# B&R Automation Studio project WithUpgradesWorking23_08_24 (part 2)

##### ams_rx_msgs.st
```iecst
ACTION msg_ams_000:
	// Status

	// AMS State
	gAMS.status.amsState.0 := ArCanReceive_0.ReceivedFrame.Data[0].0;
	gAMS.status.amsState.1 := ArCanReceive_0.ReceivedFrame.Data[0].1;
	gAMS.status.amsState.2 := ArCanReceive_0.ReceivedFrame.Data[0].2;
	gAMS.status.amsState.3 := ArCanReceive_0.ReceivedFrame.Data[0].3;
	gAMS.status.amsState.4 := ArCanReceive_0.ReceivedFrame.Data[0].4;

	gAMS.status.scEnabled  		:= (gAMS.status.amsStateName = 'SC_ENABLED') OR (gAMS.status.amsStateName = 'TS_ACTIVE') OR (gAMS.status.amsStateName = 'DRIVE');
	gAMS.status.prechargingDone := (gAMS.status.amsStateName = 'TS_ACTIVE') OR (gAMS.status.amsStateName = 'DRIVE');

	// Bank count
	gAMS.status.amsBankCount.0 := ArCanReceive_0.ReceivedFrame.Data[0].5;
	gAMS.status.amsBankCount.1 := ArCanReceive_0.ReceivedFrame.Data[0].6;
	gAMS.status.amsBankCount.2 := ArCanReceive_0.ReceivedFrame.Data[0].7;

	// Error signals
	gAMS.status.error.amsError 				:= ArCanReceive_0.ReceivedFrame.Data[1].0;
	gAMS.status.error.imdError 				:= ArCanReceive_0.ReceivedFrame.Data[1].1;
	gAMS.status.error.hvdcInterlockError 	:= ArCanReceive_0.ReceivedFrame.Data[1].2;
	gAMS.status.error.tempWarn 				:= ArCanReceive_0.ReceivedFrame.Data[1].3;
	gAMS.status.error.voltWarn 				:= ArCanReceive_0.ReceivedFrame.Data[1].4;
	gAMS.status.error.precharge 			:= ArCanReceive_0.ReceivedFrame.Data[1].5;
	gAMS.status.error.airMinus 				:= ArCanReceive_0.ReceivedFrame.Data[1].6;
	gAMS.status.error.airPlus 				:= ArCanReceive_0.ReceivedFrame.Data[1].7;

	// Data
	// gAMS.data.cellVoltageMin_CAN 	:= BYTE_TO_REAL(ArCanReceive_0.ReceivedFrame.Data[2]);
	gAMS.data.cellTempMax 			:= BYTE_TO_REAL(ArCanReceive_0.ReceivedFrame.Data[3]);
	gAMS.data.stateOfCharge 		:= BYTE_TO_REAL(ArCanReceive_0.ReceivedFrame.Data[4]);
	gAMS.status.Counter				:= BYTE_TO_USINT(ArCanReceive_0.ReceivedFrame.Data[5]);
	gAMS.status.RelayError 			:= BYTE_TO_USINT(ArCanReceive_0.ReceivedFrame.Data[6]);

END_ACTION

ACTION msg_ams_011:
	// Cell voltages

	getBankIdAndGroupId;

	//	 Group ID
	//	0	Cell [0-6]
	//	1	Cell [7-13]
	//	2 	Cell [14-20]
	//	3 	Cell [21-27]
	gAMS.status.bank[bankId].cellVoltage[groupId*7 + 0] := BYTE_TO_REAL(ArCanReceive_0.ReceivedFrame.Data[1])*0.02;
	gAMS.status.bank[bankId].cellVoltage[groupId*7 + 1] := BYTE_TO_REAL(ArCanReceive_0.ReceivedFrame.Data[2])*0.02;
	gAMS.status.bank[bankId].cellVoltage[groupId*7 + 2] := BYTE_TO_REAL(ArCanReceive_0.ReceivedFrame.Data[3])*0.02;
	gAMS.status.bank[bankId].cellVoltage[groupId*7 + 3] := BYTE_TO_REAL(ArCanReceive_0.ReceivedFrame.Data[4])*0.02;
	gAMS.status.bank[bankId].cellVoltage[groupId*7 + 4] := BYTE_TO_REAL(ArCanReceive_0.ReceivedFrame.Data[5])*0.02;
	gAMS.status.bank[bankId].cellVoltage[groupId*7 + 5] := BYTE_TO_REAL(ArCanReceive_0.ReceivedFrame.Data[6])*0.02;
	gAMS.status.bank[bankId].cellVoltage[groupId*7 + 6] := BYTE_TO_REAL(ArCanReceive_0.ReceivedFrame.Data[7])*0.02;

END_ACTION

ACTION msg_ams_012:
	// Cell temperatures

	getBankIdAndGroupId;

	// Group Id
	//	0 	Cell [0-4]
	//	1	Cell [5-9]
	gAMS.status.bank[bankId].temperatures[groupId*5 + 0] := BYTE_TO_REAL(ArCanReceive_0.ReceivedFrame.Data[1]);
	gAMS.status.bank[bankId].temperatures[groupId*5 + 1] := BYTE_TO_REAL(ArCanReceive_0.ReceivedFrame.Data[2]);
	gAMS.status.bank[bankId].temperatures[groupId*5 + 2] := BYTE_TO_REAL(ArCanReceive_0.ReceivedFrame.Data[3]);
	gAMS.status.bank[bankId].temperatures[groupId*5 + 3] := BYTE_TO_REAL(ArCanReceive_0.ReceivedFrame.Data[4]);
	gAMS.status.bank[bankId].temperatures[groupId*5 + 4] := BYTE_TO_REAL(ArCanReceive_0.ReceivedFrame.Data[5]); // Changed to 5, was 4 before? May be an error

END_ACTION

ACTION msg_ams_013:
	// Discharge Cell temperatures

	getBankIdAndGroupId;

	// Group Id
	//	0 	Cell [0-6]
	//	1	Cell [7-13]
	gAMS.status.bank[bankId].resistorTemperature[groupId*7 + 0] := BYTE_TO_REAL(ArCanReceive_0.ReceivedFrame.Data[1]);
	gAMS.status.bank[bankId].resistorTemperature[groupId*7 + 1] := BYTE_TO_REAL(ArCanReceive_0.ReceivedFrame.Data[2]);
	gAMS.status.bank[bankId].resistorTemperature[groupId*7 + 2] := BYTE_TO_REAL(ArCanReceive_0.ReceivedFrame.Data[3]);
	gAMS.status.bank[bankId].resistorTemperature[groupId*7 + 3] := BYTE_TO_REAL(ArCanReceive_0.ReceivedFrame.Data[4]);
	gAMS.status.bank[bankId].resistorTemperature[groupId*7 + 4] := BYTE_TO_REAL(ArCanReceive_0.ReceivedFrame.Data[4]);
	gAMS.status.bank[bankId].resistorTemperature[groupId*7 + 5] := BYTE_TO_REAL(ArCanReceive_0.ReceivedFrame.Data[4]);
	gAMS.status.bank[bankId].resistorTemperature[groupId*7 + 6] := BYTE_TO_REAL(ArCanReceive_0.ReceivedFrame.Data[4]);
END_ACTION

ACTION msg_ams_014:
	// Extract first byte which contains the error ID
	errorId := BYTE_TO_USINT(ArCanReceive_0.ReceivedFrame.Data[0]);

	// Reset error timer
	gAMS.status.error.errorTimers[errorId-1](IN := FALSE);
	gAMS.status.error.errorTimers[errorId-1](IN := TRUE);

	//	1  ERROR_AMS_CELL_VOLTAGE_LOW
	//	2  ERROR_AMS_CELL_VOLTAGE_HIGH
	//	3  ERROR_AMS_CELL_TEMP_LOW
	//	4  ERROR_AMS_CELL_TEMP_HIGH
	//	5  ERROR_AMS_LTC6813_COMM
	//	6  ERROR_AMS_SHUNT_COMM
	//	7  ERROR_AMS_UNABLE_TO_OPEN_SC
	//	8  ERROR_AMS_UNABLE_TO_CLOSE_SC
	//	9  ERROR_AMS_UNABLE_TO_OPEN_AIR-
	//	10 ERROR_AMS_UNABLE_TO_CLOSE_AIR-
	//	11 ERROR_AMS_UNABLE_TO_OPEN_AIR+
	//	12 ERROR_AMS_UNABLE_TO_CLOSE_AIR+
	//	13 ERROR_AMS_UNABLE_TO_OPEN_PRE+
	//	14 ERROR_AMS_UNABLE_TO_CLOSE_PRE+
	//	15 ERROR_AMS_PRE_TIMEOUT
	//	16 ERROR_AMS_UNEXPECTED_CHARGE_RATE
	//	17 ERROR_AMS_BANK_COUNT_MISMATCH
	//	18 ERROR_AMS_UNEXSPECPTED_TS_CURRENT
	//	19 ERROR_AMS_RELAY_FAIELD
	//	20 ERROR_AMS_SC_BROKEN
	//	21 AMS_UNFIT_CHARGE_VOLTAGE
	//	22 AMS_MONITOR_ERROR
END_ACTION
```

##### convertData.st
```iecst
ACTION convertData:
	// Takes in data in big endian and converts it to data in litte endian (which is used by the PLC)
	// Switch endian
	dataArr[3] := ArCanReceive_0.ReceivedFrame.Data[2];
	dataArr[2] := ArCanReceive_0.ReceivedFrame.Data[3];
	dataArr[1] := ArCanReceive_0.ReceivedFrame.Data[4];
	dataArr[0] := ArCanReceive_0.ReceivedFrame.Data[5];
	// Extract data from array
	memcpy(ADR(data), ADR(dataArr),4);
END_ACTION
```

##### orion_rx_msgs.st
```iecst
// Frame ID's correspoinding to the orion bms
//  Some message
ACTION msg_orion_001:
	// Byte 0 and 1
	brsmemcpy(ADR(packPower), ADR(ArCanReceive_0.ReceivedFrame.Data[0]), 2 * SIZEOF(ArCanReceive_0.ReceivedFrame.Data[0]));
	gORION.data.packPower 	:= INT_TO_REAL(packPower) / 10; // packpower sent as 0.1kW
	gAMS.data.packPower 	:= gORION.data.packPower;

	// byte 2 and 3, Total pack voltage
	brsmemcpy(ADR(packVoltage), ADR(ArCanReceive_0.ReceivedFrame.Data[2]), 2 * SIZEOF(ArCanReceive_0.ReceivedFrame.Data[2]));
	gAMS.data.batteryVoltage 	:= UINT_TO_REAL(packVoltage) / 10; // Pack voltage sent as 0.1V
	gORION.data.packVoltage 	:= gAMS.data.batteryVoltage;

	// Byte 4 and 5, Total pack Current
	brsmemcpy(ADR(packCurrent), ADR(ArCanReceive_0.ReceivedFrame.Data[4]), 2 * SIZEOF(ArCanReceive_0.ReceivedFrame.Data[4]));
	gAMS.data.outputCurrent 	:= INT_TO_REAL(packCurrent) / 10; // Pack Current sent as 0.1A
	gORION.data.outputCurrent 	:= gAMS.data.outputCurrent;
	gORION.data.chargeCurrent	:= - gAMS.data.outputCurrent;

	// Byte 6 and 7, Charge Current Limit
	brsmemcpy(ADR(gORION.data.CCL), ADR(ArCanReceive_0.ReceivedFrame.Data[6]), 2 * SIZEOF(ArCanReceive_0.ReceivedFrame.Data[6]));

END_ACTION

// Errors and DTC STATUS
ACTION msg_orion_002:
	// BYte 0 and 1
	brsmemcpy(ADR(gAMS.status.DTC1Status), ADR(ArCanReceive_0.ReceivedFrame.Data[0]), 2* SIZEOF(ArCanReceive_0.ReceivedFrame.Data[0]));
	// Byte 2 and 3
	brsmemcpy(ADR(gAMS.status.DTC2Status), ADR(ArCanReceive_0.ReceivedFrame.Data[2]), 2* SIZEOF(ArCanReceive_0.ReceivedFrame.Data[2]));
	gAMS.status.error.highVoltage	:= gAMS.status.DTC1Status.5 OR gAMS.status.DTC2Status.6;
	gAMS.status.error.lowVoltage	:= gAMS.status.DTC1Status.6 OR gAMS.status.DTC2Status.6;
	gAMS.status.error.highTemp 		:= gAMS.status.DTC1Status.7;

	// Byte 4
	// Make some flag wih the MPI to tell the status of these
	gAMS.status.error.imdError 		:= ArCanReceive_0.ReceivedFrame.Data[4].0;
	gAMS.status.error.amsError 		:= ArCanReceive_0.ReceivedFrame.Data[4].1;
	//gAMS.status.error.openSc		:= ArCanReceive_0.ReceivedFrame.Data[4].2;
	gAMS.status.scEnabled			:= ArCanReceive_0.ReceivedFrame.Data[4].2;
	gORION.status.sdcEnabled		:= gAMS.status.scEnabled;
	gAMS.status.relayState.MPEnableSignalStatus := ArCanReceive_0.ReceivedFrame.Data[4].3;

	// BYte 5, rolling counter incrementing every 100ms.
	gORION.data.rollingCounter := BYTE_TO_USINT(ArCanReceive_0.ReceivedFrame.Data[5]);

	// Byte 6 and 7, Discharge Current Limit
	brsmemcpy(ADR(gORION.data.DCL), ADR(ArCanReceive_0.ReceivedFrame.Data[6]), 2 * SIZEOF(ArCanReceive_0.ReceivedFrame.Data[6]));

END_ACTION

ACTION msg_orion_003:
	// 0 and 1, state of relays (Should be sent as little endian)
	brsmemcpy(ADR(gAMS.status.relayState.relayState),ADR(ArCanReceive_0.ReceivedFrame.Data[0]), 2* SIZEOF(ArCanReceive_0.ReceivedFrame.Data[0]));
	gAMS.status.relayState.dischargeRelayEnabled 		:= gAMS.status.relayState.relayState.0;
	gAMS.status.relayState.chargeRelayEnabled	 		:= gAMS.status.relayState.relayState.1;
	gAMS.status.relayState.chargerSafetyEnabled	 		:= gAMS.status.relayState.relayState.2;
	gAMS.status.relayState.malfunctionIndicatorActive 	:= gAMS.status.relayState.relayState.3;
	gAMS.status.relayState.MPI1SignalStatus 			:= gAMS.status.relayState.relayState.4;
	gAMS.status.relayState.alwaysOnSignalStatus 		:= gAMS.status.relayState.relayState.5;
	gAMS.status.relayState.isReadyInputStatus 			:= gAMS.status.relayState.relayState.6;
	gAMS.status.relayState.isChargingInputStatus 		:= gAMS.status.relayState.relayState.7;

	// gAMS.status.relayState.MPI2SignalStatus 			:= gAMS.status.relayState.relayState.8;
	// gAMS.status.relayState.MPI3SignalStatus  		:= gAMS.status.relayState.relayState.9;
	// gAMS.status.relayState.chargeModeStatus 			:= gAMS.status.relayState.relayState.10;
	// gAMS.status.relayState.MPO2SignalStatus 			:= gAMS.status.relayState.relayState.11;
	// gAMS.status.relayState.MPO3SignalStatus 			:= gAMS.status.relayState.relayState.12;
	// gAMS.status.relayState.MPO4SignalStatus 			:= gAMS.status.relayState.relayState.13;
	// gAMS.status.relayState.MPEnableSignalStatus 		:= gAMS.status.relayState.relayState.14;
	// gAMS.status.relayState.MPO1SignalStatus 			:= gAMS.status.relayState.relayState.15;

	// byte 3
	gAMS.data.cellTempMax := BYTE_TO_REAL(ArCanReceive_0.ReceivedFrame.Data[3]); // Max cell temperature of pack, send as (1 degree celcius)
	// Since it is not possible to get all cell voltages independently, max temp i applied to all cells in logic
	appendTemps;

	// Byte 4
	gAMS.data.stateOfCharge := BYTE_TO_REAL(ArCanReceive_0.ReceivedFrame.Data[4]) / 2; // State of charge of battery, (0,5%)

	// Byte 5
	gAMS.status.Counter := BYTE_TO_USINT(ArCanReceive_0.ReceivedFrame.Data[5]); // Counter can be used to make sure Orion BMS is still running and is not stuck

	// byte 6 and 7
	// Failsafe statuses:
	brsmemcpy(ADR(gAMS.status.failsafeStatus.failsafeStatus), ADR(ArCanReceive_0.ReceivedFrame.Data[6]), 2 * SIZEOF(ArCanReceive_0.ReceivedFrame.Data[6]));
	gAMS.status.error.relayFailed := gAMS.status.failsafeStatus.failsafeStatus.2;

END_ACTION

// Related to DCL and CCL in KW
ACTION msg_orion_004:
	// Byte 0-1 Discharge Current limit expressed in KW
	brsmemcpy(ADR(DCL_KW_Temp),ADR(ArCanReceive_0.ReceivedFrame.Data[0]), 2* SIZEOF(ArCanReceive_0.ReceivedFrame.Data[0]));
	gORION.data.DCL_KW := INT_TO_REAL(DCL_KW_Temp)/10; // [0.1kW]

	// Byte 2-3 Charge Current limit expressed in KW
	brsmemcpy(ADR(CCL_KW_Temp),ADR(ArCanReceive_0.ReceivedFrame.Data[2]), 2* SIZEOF(ArCanReceive_0.ReceivedFrame.Data[2]));
	gORION.data.CCL_KW := INT_TO_REAL(CCL_KW_Temp)/10; // [0.1kW]
END_ACTION

 // CELL VOLTAGES, sent though boradcasting
ACTION msg_orion_010:

	// Broadcasted cell voltages from the orion bms
	checksumGiven 		:= BYTE_TO_USINT(ArCanReceive_0.ReceivedFrame.Data[7]);
	checksumCalculated 	:= RX_ORION_ID_BASE + 16#010 + 8;
	checksumCalculated  := checksumCalculated + BYTE_TO_UDINT(ArCanReceive_0.ReceivedFrame.Data[0]);
	checksumCalculated  := checksumCalculated + BYTE_TO_UDINT(ArCanReceive_0.ReceivedFrame.Data[1]);
	checksumCalculated  := checksumCalculated + BYTE_TO_UDINT(ArCanReceive_0.ReceivedFrame.Data[2]);
	checksumCalculated  := checksumCalculated + BYTE_TO_UDINT(ArCanReceive_0.ReceivedFrame.Data[3]);
	checksumCalculated  := checksumCalculated + BYTE_TO_UDINT(ArCanReceive_0.ReceivedFrame.Data[4]);
	checksumCalculated  := checksumCalculated + BYTE_TO_UDINT(ArCanReceive_0.ReceivedFrame.Data[5]);
	checksumCalculated  := checksumCalculated + BYTE_TO_UDINT(ArCanReceive_0.ReceivedFrame.Data[6]);

	brsmemcpy(ADR(checksumValidate),ADR(checksumCalculated),1);

	// Checking if checksum is good
	IF checksumGiven = checksumValidate THEN
		checksumCorrect := checksumCorrect +1;
		// The checksum is correct and data is overwritten
		cellId := BYTE_TO_USINT(ArCanReceive_0.ReceivedFrame.Data[0]);
		brsmemcpy(ADR(tempVoltageHigh), ADR(ArCanReceive_0.ReceivedFrame.Data[1]), SIZEOF(ArCanReceive_0.ReceivedFrame.Data[1]));
		brsmemcpy(ADR(tempVoltageLow), ADR(ArCanReceive_0.ReceivedFrame.Data[2]), SIZEOF(ArCanReceive_0.ReceivedFrame.Data[2]));
		tempVoltage := tempVoltageLow + 256 * tempVoltageHigh;
		gAMS.status.pack.InstantCellVoltage[cellId] := (UINT_TO_REAL(tempVoltage)) / 10000; // recieved data is 2 byte, 0.1mV

		brsmemcpy(ADR(tempVoltageHigh), ADR(ArCanReceive_0.ReceivedFrame.Data[5]), SIZEOF(ArCanReceive_0.ReceivedFrame.Data[5]));
		brsmemcpy(ADR(tempVoltageLow), ADR(ArCanReceive_0.ReceivedFrame.Data[6]), SIZEOF(ArCanReceive_0.ReceivedFrame.Data[6]));
		tempVoltage := tempVoltageLow + 256 * tempVoltageHigh;
		gAMS.status.pack.cellVoltage[cellId] 		:= (UINT_TO_REAL(tempVoltage)) / 10000; // recieved data is 2 byte, 0.1mV

		cellidToBankAndCell;
		gAMS.status.bank[bankId].cellVoltage[bankCellId] := gAMS.status.pack.cellVoltage[cellId];
	END_IF;

END_ACTION

// CELL TEMPERATURES
ACTION msg_orion_011:
	// Broadcasted cell temperatures from the orion bms
	// Is not currently possible to implement
END_ACTION
```

##### shunt_rx_msgs.st
```iecst
ACTION msg_shunt_021:

	// Check if message is of type 'Result' which means it contains measured data and not configuration data
	// If byte 0 is b'0000xxxx' (the 4 msb's are 0) then the type of 'Result'
	IF ArCanReceive_0.ReceivedFrame.Data[0].7 = 0 AND ArCanReceive_0.ReceivedFrame.Data[0].6 = 0 AND
		ArCanReceive_0.ReceivedFrame.Data[0].5 = 0 AND ArCanReceive_0.ReceivedFrame.Data[0].4 = 0 THEN
		// Extract data and switch from big to little endian
		convertData;
		gShunt.data.actCurrent := UDINT_TO_REAL(data)/1000.0; // sent as big indian 4 bytes. [1mA]
	END_IF;

END_ACTION

//Considered to be voltage of the TS side of the car
ACTION msg_shunt_022:
	IF ArCanReceive_0.ReceivedFrame.Data[0].7 = 0 AND ArCanReceive_0.ReceivedFrame.Data[0].6 = 0 AND
		ArCanReceive_0.ReceivedFrame.Data[0].5 = 0 AND ArCanReceive_0.ReceivedFrame.Data[0].4 = 0 THEN
		// Extract data
		convertData;
		gShunt.data.actVoltage := UDINT_TO_REAL(data)/1000.0; // sent as big indian 4 bytes. [1mV]
	END_IF;

END_ACTION

// Not currently in use
ACTION msg_shunt_023:
	IF ArCanReceive_0.ReceivedFrame.Data[0].7 = 0 AND ArCanReceive_0.ReceivedFrame.Data[0].6 = 0 AND
		ArCanReceive_0.ReceivedFrame.Data[0].5 = 0 AND ArCanReceive_0.ReceivedFrame.Data[0].4 = 0 THEN
		// Extract data
		convertData;
		gShunt.data.actVoltage2 := UDINT_TO_REAL(data)/1000.0; // sent as big indian 4 bytes. [1mV]
	END_IF;
END_ACTION

ACTION msg_shunt_026:
	IF ArCanReceive_0.ReceivedFrame.Data[0].7 = 0 AND ArCanReceive_0.ReceivedFrame.Data[0].6 = 0 AND
		ArCanReceive_0.ReceivedFrame.Data[0].5 = 0 AND ArCanReceive_0.ReceivedFrame.Data[0].4 = 0 THEN
		// Extract data
		convertData;
		gShunt.data.actPowerW := UDINT_TO_REAL(data);
		gShunt.data.actPowerKW := gShunt.data.actPowerW/1000.0; // sent as big indian 4 bytes. [1mW]
	END_IF;
END_ACTION

ACTION msg_shunt_027:
	IF ArCanReceive_0.ReceivedFrame.Data[0].7 = 0 AND ArCanReceive_0.ReceivedFrame.Data[0].6 = 0 AND
		ArCanReceive_0.ReceivedFrame.Data[0].5 = 0 AND ArCanReceive_0.ReceivedFrame.Data[0].4 = 0 THEN
		// Extract data
		convertData;
		gShunt.data.actCurrentAS := UDINT_TO_REAL(data);
	END_IF;
END_ACTION

ACTION msg_shunt_028:
	IF ArCanReceive_0.ReceivedFrame.Data[0].7 = 0 AND ArCanReceive_0.ReceivedFrame.Data[0].6 = 0 AND
		ArCanReceive_0.ReceivedFrame.Data[0].5 = 0 AND ArCanReceive_0.ReceivedFrame.Data[0].4 = 0 THEN
		// Extract data
		convertData;
		gShunt.data.actPowerWH  := UDINT_TO_REAL(data);
		gShunt.data.actPowerKWH := gShunt.data.actPowerWH/1000.0;
	END_IF;
END_ACTION
```

### globalDashboard.typ
```iecst
TYPE
	gDashboard_typ : 	STRUCT
		status : gDashboard_status_typ;
		inputs : gDashboard_inputs_typ;
		outputs : gDashboard_outputs_typ;
		cmd : gDashboard_cmd_typ;
		data : gDashboard_data_typ;
	END_STRUCT;
	gDashboard_status_typ : 	STRUCT
		ok : BOOL;
		DashboardDisconnected : BOOL;
		unknownMessageReceived : BOOL;
		unknownMessageID : UDINT;
		timeoutFromDashboard : BOOL;
		canFramesLost : BOOL;
		statusIndex : USINT;
		errorCode : USINT;
	END_STRUCT;
	gDashboard_data_typ : 	STRUCT
		dummy : USINT;
	END_STRUCT;
	gDashboard_inputs_typ : 	STRUCT
		di_buttonSafety : BOOL;
		di_buttonTractive : BOOL;
		di_buttonDrive : BOOL;
		di_button1 : BOOL;
		di_button2 : BOOL;
		di_button3 : BOOL;
		di_button4 : BOOL;
	END_STRUCT;
	gDashboard_cmd_typ : 	STRUCT
		sendVehicleConfigMsg : BOOL;
	END_STRUCT;
	gDashboard_outputs_typ : 	STRUCT
		do_ledTS_OFF : BOOL;
		do_ledIMD : BOOL;
		do_ledAMS : BOOL;
		do_ledEBS : BOOL;
		do_ledREADY : USINT;
		do_ledSC : USINT;
		do_ledLV : BOOL;
		do_ledDV : BOOL;
		Error : USINT;
		com_error_SC : BOOL;
		com_error_Shunt : BOOL;
		com_error_AMS : BOOL;
		com_error_Datalog : BOOL;
		com_error_Dashboard : BOOL;
		com_error_3rd_Inv : BOOL;
		com_error_2nd_Inv : BOOL;
		com_error_1st_Inv : BOOL;
		com_error_0_Inv : BOOL;
		com_error_INS : BOOL;
		com_error_SteeringAngle : BOOL;
		com_error_BreakPressure_Front : BOOL;
		com_error_BreakPressure_Back : BOOL;
		com_error_TorquePedal : BOOL;
		com_error_TorquePedal_Plausi : BOOL;
		com_error_RTDS : BOOL;
		com_error_Cooling : BOOL;
		com_error_LV : BOOL;
		com_error_HighTemperature : BOOL;
	END_STRUCT;
END_TYPE
```

### Program Logical/Dashboard/Dashboard (IEC)

#### Types.typ - Local data types
```iecst
TYPE
	led_states :
		(
		ON,
		OFF,
		BLINKING
		);
END_TYPE
```

#### Variables.var - Local variables
```iecst
VAR
	ledLVState : USINT;
	scLedState : led_states;
	estimatedRange : UINT;
	msgIndex : USINT;
	i : USINT;
	speed : UINT;
	soc : UINT;
	maxTemperature : UINT;
	lvBatVoltage : UINT;
	torqueLimitNm : UINT;
	powerLimitKW : UINT;
	TON_sc : TON;
	ArCanSetBaudrate_0 : ArCanSetBaudrate;
	ArCanSend_0 : ArCanSend;
	ArCanReceive_0 : ArCanReceive;
	communicationState : CAN_STATES;
	deviceName : STRING[127];
	TON_disconnectTimer : TON;
	TON_sendTimer : TON;
	frameIdOffset : UDINT;
	TX_CAN_ID_BASE : {REDUND_UNREPLICABLE} UDINT := 0;
	RX_CAN_ID_BASE : {REDUND_UNREPLICABLE} UDINT := 0;
END_VAR
VAR CONSTANT
	READY_OFF : USINT := 0;
	READY_ON : USINT := 1;
	READY_SLOW_BLINK : USINT := 2;
	READY_FAST_BLINK : USINT := 3;
	SC_OFF : USINT := 0;
	SC_ON : USINT := 1;
	SC_BLINK : USINT := 2;
END_VAR
```

#### ledAMS.st
```iecst
(* Control the AMS LED *)
ACTION ledAMS:
	IF gStateMachine.status.state = STATE_INITIALIZE THEN
		gDashboard.outputs.do_ledAMS := TRUE;
	ELSE
		gDashboard.outputs.do_ledAMS := gAMS.status.error.amsError;
	END_IF;

END_ACTION
```

#### ledSC.st
```iecst
(* Control the SC LED *)

ACTION ledSC:

 	IF gStateMachine.status.state = STATE_INITIALIZE THEN
		gDashboard.outputs.do_ledSC := SC_ON;
	ELSE
		IF gSafetyChain.status.scOK_notEnabled = TRUE AND gSafetyChain.status.scOK = FALSE THEN // If safety chain is OK, but enable button is false change to BLINKING
			gDashboard.outputs.do_ledSC := SC_BLINK;
		ELSIF gSafetyChain.status.scOK = TRUE THEN
			gDashboard.outputs.do_ledSC := SC_ON;
		ELSE
			gDashboard.outputs.do_ledSC := SC_OFF;
		END_IF
	END_IF

END_ACTION
```

#### Send_Bus.st
```iecst
ACTION Send_Bus:

	(* Set timer *)
	TON_sendTimer.PT := T#100ms;
//	TON_sendTimer.PT := T#25ms;

	(* If timer runs out *)
	IF NOT gIsSimulation THEN
		IF TON_sendTimer.Q THEN
			(* Go through each message. Encode and send them *)
			//			FOR i := 0 TO 3 DO
				CASE msgIndex OF
					0: msg_0x000;
					1: msg_0x001;
					2: msg_0x002;
					3: msg_0x003;
					4: msg_0x004;
					ELSE
				END_CASE;
			ArCanSend_0(SendFrame := TRUE);
			ArCanSend_0(SendFrame := FALSE);

			msgIndex := msgIndex + 1;
			IF msgIndex > 4 THEN
				msgIndex := 0;
			END_IF;

//			END_FOR;
			(* Reset timer *)
			TON_sendTimer(IN:=FALSE);
		END_IF;

//		IF gDashboard.cmd.sendVehicleConfigMsg THEN
//			gDashboard.cmd.sendVehicleConfigMsg := FALSE;
//			msg_0x003;
//			ArCanSend_0(SendFrame := TRUE);
//			ArCanSend_0(SendFrame := FALSE);
//		END_IF;

	END_IF;

	(* Start timer *)
	TON_sendTimer(IN:=TRUE);

	ArCanSend_0();
END_ACTION
```

### globalTorqueSensor.typ
```iecst
TYPE
	gTorqueSensor_cmd_typ : 	STRUCT
		torque1 : INT;
		torque2 : INT;
		disablePlausibilityCheck : BOOL;
	END_STRUCT;
	gTorqueSensor_typ : 	STRUCT
		status : gTorqueSensor_status_typ;
		inputs : gTorqueSensor_inputs_typ;
		outputs : gTorqueSensor_outputs_typ;
		data : gTorqueSensor_data_typ;
		cmd : gTorqueSensor_cmd_typ;
	END_STRUCT;
	gTorqueSensor_status_typ : 	STRUCT
		ok : BOOL;
		errorOutOfRangeSensor1 : BOOL;
		errorOutOfRangeSensor2 : BOOL;
		plausibilityError : BOOL;
		torqueEnabled : BOOL;
		torquePercentage : REAL;
		criticalError : BOOL;
		maxTorquePercent : USINT;
	END_STRUCT;
	gTorqueSensor_data_typ : 	STRUCT
		torque1Percent : REAL;
		torque2Percent : REAL;
	END_STRUCT;
	gTorqueSensor_inputs_typ : 	STRUCT
		torque1 : INT;
		torque2 : INT;
	END_STRUCT;
	gTorqueSensor_outputs_typ : 	STRUCT
		dummy : USINT;
	END_STRUCT;
END_TYPE
```

### globalLowVoltageBattery.typ
```iecst
TYPE
	gLowVoltageBattery_typ : 	STRUCT
		status : gLowVoltageBattery_status_typ;
		inputs : gLowVoltageBattery_inputs_typ;
		outputs : gLowVoltageBattery_outputs_typ;
		data : gLowVoltageBattery_data_typ;
	END_STRUCT;
	gLowVoltageBattery_status_typ : 	STRUCT
		full : BOOL;
		empty : BOOL;
		percentageSoc : REAL;
	END_STRUCT;
	gLowVoltageBattery_data_typ : 	STRUCT
		current : REAL;
		voltage : REAL;
	END_STRUCT;
	gLowVoltageBattery_inputs_typ : 	STRUCT
		ai_current : INT;
		ai_voltage : INT;
	END_STRUCT;
	gLowVoltageBattery_outputs_typ : 	STRUCT
		dummy : USINT;
	END_STRUCT;
END_TYPE
```

### globalLowVoltageBattery.var
```iecst
VAR
	gLowVoltageBattery : gLowVoltageBattery_typ;
END_VAR
```

### Program Logical/Sensors/Sensors (IEC)

#### Types.typ - Local data types
```iecst
TYPE
	braking_pedal_variables_typ : 	STRUCT
		brakingPedalFrontMax : UINT;
		brakingPedalFrontMin : UINT;
		brakingPedalRearMax : UINT;
		brakingPedalRearMin : UINT;
		slope : REAL;
	END_STRUCT;
	braking_pedal_constants_typ : 	STRUCT
		frontWarningLimitMaxMax : UINT;
		frontWarningLimitMax : UINT;
		frontWarningLimitMin : UINT;
		frontWarningLimitMinMin : UINT;
		rearWarningLimitMaxMax : UINT;
		rearWarningLimitMax : UINT;
		rearWarningLimitMin : UINT;
		rearWarningLimitMinMin : UINT;
		softBrakingLimit : UINT;
		hardBrakingLimit : UINT;
	END_STRUCT;
	torque_pedal_variables_typ : 	STRUCT
		torquePedalMax2 : UINT;
		torquePedalMax1 : UINT;
		torquePedalMin2 : UINT;
		torquePedalMin1 : UINT;
		TON_torqueOff : TON;
		slope : REAL;
	END_STRUCT;
	torque_pedal_constants_typ : 	STRUCT
		lowLimit2 : UINT;
		highLimit2 : UINT;
		lowLimit1 : UINT;
		highLimit1 : UINT;
		torqueOffUpperHysteresis : REAL;
		torqueOffLowerHysteresis : REAL;
	END_STRUCT;
	steering_angle_constants_typ : 	STRUCT
		highLimit : UINT;
		lowLimit : UINT;
		disconnectionLimit : UINT;
		MAX_ANGLE : REAL;
		MIN_ANGLE : REAL;
	END_STRUCT;
	steering_angle_variables_typ : 	STRUCT
		steeringWheelAngleStr : STRING[80];
		wheelAngleStr : STRING[80];
		leftValue : UINT;
		rightValue : UINT;
	END_STRUCT;
	lv_battery_constants_typ : 	STRUCT
		HighLimit : REAL;
		LowLimit : REAL;
	END_STRUCT;
	lv_battery_variable_typ : 	STRUCT
		TON_batteryEmpty : TON;
		TON_batteryFull : TON;
	END_STRUCT;
END_TYPE
```

#### BrakingPedal.st
```iecst
ACTION BrakingPedalInit:
	(* Sensor limit values *)
	brakingPedalVariables.brakingPedalRearMax 		:= 8000;
	brakingPedalVariables.brakingPedalRearMin 		:= 1655;
	brakingPedalVariables.brakingPedalFrontMax 		:= 8000;
	brakingPedalVariables.brakingPedalFrontMin 		:= 1655;

	(* Braking limits *)
	brakingPedalConstants.hardBrakingLimit			:= 5400;
	brakingPedalConstants.softBrakingLimit			:= 2000;

	(* Upper limit symboling an electrical fault *)
//	brakingPedalConstants.frontWarningLimitMaxMax 	:= brakingPedalVariables.brakingPedalFrontMax + 500;
//	brakingPedalConstants.rearWarningLimitMaxMax 	:= brakingPedalVariables.brakingPedalRearMax  + 500;
	brakingPedalConstants.frontWarningLimitMaxMax 	:= 15250;
	brakingPedalConstants.rearWarningLimitMaxMax 	:= 15250;

	(* Upper limit symboling a mechanical fault *)
	brakingPedalConstants.frontWarningLimitMax 		:= brakingPedalVariables.brakingPedalFrontMax + 100;
	brakingPedalConstants.rearWarningLimitMax 		:= brakingPedalVariables.brakingPedalRearMax  + 100;

	(* Lower limit symboling a mechanical fault *)
	brakingPedalConstants.frontWarningLimitMin 		:= brakingPedalVariables.brakingPedalFrontMin - 100;
	brakingPedalConstants.rearWarningLimitMin 		:= brakingPedalVariables.brakingPedalRearMin  - 100;

	(* Lower limit symboling an electrical fault *)
	brakingPedalConstants.frontWarningLimitMinMin 	:= brakingPedalVariables.brakingPedalFrontMin - 500;
	brakingPedalConstants.rearWarningLimitMinMin 	:= brakingPedalVariables.brakingPedalRearMin  - 500;

END_ACTION

ACTION BrakingPedal:
	(* Detect if brake pedal is being pressed lightly *)
	gBraking.status.softBraking 		 := INT_TO_UINT(gBraking.inputs.ai_brakePressureFront) > brakingPedalConstants.softBrakingLimit OR
											INT_TO_UINT(gBraking.inputs.ai_brakePressureRear)  > brakingPedalConstants.softBrakingLimit OR
											gSoftBrakingForced;

	(* Detect hard braking *)
	gBraking.status.hardBraking 		 := INT_TO_UINT(gBraking.inputs.ai_brakePressureFront) > brakingPedalConstants.hardBrakingLimit OR
										    INT_TO_UINT(gBraking.inputs.ai_brakePressureRear)  > brakingPedalConstants.hardBrakingLimit;

	(* Control brakelight *)
	IF gStateMachine.status.state <> STATE_INITIALIZE THEN
		gBraking.outputs.do_brakeLight   := gBraking.status.softBraking;
	END_IF

	(* Check if brake pressures are out of range *)
	// If brake pressure front get above limit, an error message is shown.
	gBraking.status.errorOutOfRangeFront := INT_TO_UINT(gBraking.inputs.ai_brakePressureFront) >= brakingPedalConstants.frontWarningLimitMax OR
											INT_TO_UINT(gBraking.inputs.ai_brakePressureFront) <= brakingPedalConstants.frontWarningLimitMin;

	// If brake pressure rear get above limit, an error message is shown.
	gBraking.status.errorOutOfRangeRear := 	INT_TO_UINT(gBraking.inputs.ai_brakePressureRear) >= brakingPedalConstants.rearWarningLimitMax OR
											INT_TO_UINT(gBraking.inputs.ai_brakePressureRear) <= brakingPedalConstants.rearWarningLimitMin;

	(* Calculate pedal percentages *)
	IF NOT gBraking.status.errorOutOfRangeFront THEN
		brakingPedalVariables.slope := (100.00)/(UINT_TO_REAL(brakingPedalVariables.brakingPedalFrontMax) - UINT_TO_REAL(brakingPedalVariables.brakingPedalFrontMin));
		gBraking.data.pressurePercentageFront := LIMIT(0 ,brakingPedalVariables.slope * (INT_TO_REAL(gBraking.inputs.ai_brakePressureFront)-UINT_TO_REAL(brakingPedalVariables.brakingPedalFrontMin)),100);
	ELSE
		gBraking.data.pressurePercentageFront := 0;
	END_IF;

	IF NOT gBraking.status.errorOutOfRangeRear THEN
		brakingPedalVariables.slope := (100.00)/(UINT_TO_REAL(brakingPedalVariables.brakingPedalRearMax) - UINT_TO_REAL(brakingPedalVariables.brakingPedalRearMin));
		gBraking.data.pressurePercentageRear := LIMIT(0 ,brakingPedalVariables.slope * (INT_TO_REAL(gBraking.inputs.ai_brakePressureRear)-UINT_TO_REAL(brakingPedalVariables.brakingPedalRearMin)),100);
	ELSE
		gBraking.data.pressurePercentageRear := 0;
	END_IF;

	gBraking.data.pressurePercentage := (gBraking.data.pressurePercentageFront + gBraking.data.pressurePercentageRear)/2.0;

	(* Determine if the brake pedal + sensors are working properly *)
	gBraking.status.ok := NOT gBraking.status.errorOutOfRangeFront AND NOT gBraking.status.errorOutOfRangeRear;

	// Calculate actual pressure
	gBraking.data.pressureBarFront 	:= ((INT_TO_REAL(gBraking.inputs.ai_brakePressureFront)*10/32768)-0.5)*40;
	gBraking.data.pressureBarRear	:= ((INT_TO_REAL(gBraking.inputs.ai_brakePressureRear)*10/32768)-0.5)*40;

END_ACTION
```

#### TorquePedal.st
```iecst
ACTION TorquePedalInit:
	(* Sensor edge values *)
	torquePedalVariables.torquePedalMin1 	:= 13636;
	torquePedalVariables.torquePedalMin2 	:= 2415;
	torquePedalVariables.torquePedalMax1 	:= 21181;
	torquePedalVariables.torquePedalMax2 	:= 7947;

	// Constant for limit torque percent
	IF maxTorquePercentThrottle = 0 THEN
		maxTorquePercentThrottle := 50; // Change to 100, Max Torque Percent
	END_IF;
	gTorqueSensor.status.maxTorquePercent := maxTorquePercentThrottle;

	(* Range for torque sensor 1 *)
	torquePedalConstants.highLimit1 := torquePedalVariables.torquePedalMax1 + 200;
	torquePedalConstants.lowLimit1  := 0;

	(* Range for torque sensor 2 *)
	torquePedalConstants.highLimit2 := torquePedalVariables.torquePedalMax2 + 200;
	torquePedalConstants.lowLimit2 	:= 0;

	(* Torque off hysteresis values *)
	torquePedalConstants.torqueOffUpperHysteresis := 25; // [%]
	torquePedalConstants.torqueOffLowerHysteresis := 5;  // [%]

	(* Plausibility check disable (for test setup) *)
	gTorqueSensor.cmd.disablePlausibilityCheck := FALSE;
END_ACTION

ACTION TorquePedal:
	// Percent of MAX torque at full throttle:
	gTorqueSensor.status.maxTorquePercent := maxTorquePercentThrottle;

	gTorqueSensor.status.errorOutOfRangeSensor1 := 	INT_TO_UINT(gTorqueSensor.inputs.torque1) > torquePedalConstants.highLimit1 OR
													INT_TO_UINT(gTorqueSensor.inputs.torque1) < torquePedalConstants.lowLimit1;

	gTorqueSensor.status.errorOutOfRangeSensor2 := 	INT_TO_UINT(gTorqueSensor.inputs.torque2) > torquePedalConstants.highLimit2 OR
													INT_TO_UINT(gTorqueSensor.inputs.torque2) < torquePedalConstants.lowLimit2;

	(* Calculate pedal percentages *)

	// Sensor 1
	IF NOT gTorqueSensor.status.errorOutOfRangeSensor1 THEN
		torquePedalVariables.slope := (100)/(UINT_TO_REAL(torquePedalVariables.torquePedalMax1) - UINT_TO_REAL(torquePedalVariables.torquePedalMin1));
		gTorqueSensor.data.torque1Percent := LIMIT(0 ,torquePedalVariables.slope * (INT_TO_REAL(gTorqueSensor.inputs.torque1)-(10+UINT_TO_REAL(torquePedalVariables.torquePedalMin1))),100);
	ELSE
		gTorqueSensor.data.torque1Percent := 0;
	END_IF;
	// gTorqueSensor.status.maxTorquePercent TODO: USE THIS FOR SCALING
	// Sensor 2
	IF NOT gTorqueSensor.status.errorOutOfRangeSensor2 THEN
		torquePedalVariables.slope := (100)/(UINT_TO_REAL(torquePedalVariables.torquePedalMax2) - UINT_TO_REAL(torquePedalVariables.torquePedalMin2));
		gTorqueSensor.data.torque2Percent := LIMIT(0 ,torquePedalVariables.slope * (INT_TO_REAL(gTorqueSensor.inputs.torque2)-UINT_TO_REAL(torquePedalVariables.torquePedalMin2)),100);
	ELSE
		gTorqueSensor.data.torque2Percent := 0;
	END_IF;

	// Sensor 1 is arbitrarily taken to be the torque percentage
	// Value is then scaled by desired power
	gTorqueSensor.status.torquePercentage := gTorqueSensor.data.torque1Percent*gTorqueSensor.status.maxTorquePercent/100;

	(* Test if torque sensor values are out of range of each other*)
	TorqueSensorsOutOfRange;
	TorqueOff;

	(* Report critical error if either of the torque pedal sensors leave their working range *)
	gTorqueSensor.status.criticalError := gTorqueSensor.status.errorOutOfRangeSensor1 OR gTorqueSensor.status.errorOutOfRangeSensor2 OR gTorqueSensor.status.plausibilityError;

	(* Determine if the torque pedal is working properly *)
	gTorqueSensor.status.ok := NOT gTorqueSensor.status.criticalError;

END_ACTION

(* Test if torque pedals are more than 10% different than each other *)
ACTION TorqueSensorsOutOfRange:
	IF gTorqueSensor.cmd.disablePlausibilityCheck THEN
		gTorqueSensor.status.plausibilityError := FALSE;
	ELSE
		// check if torque sensor 1 and 2 vary more than 5 %
		gTorqueSensor.status.plausibilityError := ABS(gTorqueSensor.data.torque1Percent - gTorqueSensor.data.torque2Percent) > 5;
	END_IF;
END_ACTION

ACTION TorqueOff:
	IF gTorqueSensor.status.torqueEnabled THEN
		(* Test the criterias for turning off the torque. If they are met start timer *)
		IF 	gBraking.status.softBraking AND
			(gTorqueSensor.data.torque1Percent >= torquePedalConstants.torqueOffUpperHysteresis OR
			 gTorqueSensor.data.torque2Percent >= torquePedalConstants.torqueOffUpperHysteresis OR
		 	 gORION.data.packPower >= 5.0) THEN

			torquePedalVariables.TON_torqueOff.PT := T#250ms;	// Set timer duration TODO: Change to 500 that is the limit in the rules
			torquePedalVariables.TON_torqueOff.IN := TRUE;		// Start timer
		ELSE
			torquePedalVariables.TON_torqueOff.IN := FALSE;		// Else stop timer
		END_IF

		IF torquePedalVariables.TON_torqueOff.Q THEN			// If timer runs out
			gTorqueSensor.status.torqueEnabled := FALSE;		// Remove torque
		ELSE
			gTorqueSensor.status.torqueEnabled := TRUE;			// Else keep torque
		END_IF;
	ELSE
		(* Test the criterias for turning on the torque *)
		gTorqueSensor.status.torqueEnabled := 	gTorqueSensor.data.torque1Percent < torquePedalConstants.torqueOffLowerHysteresis AND
												gTorqueSensor.data.torque2Percent < torquePedalConstants.torqueOffLowerHysteresis AND (NOT gBraking.status.softBraking);
		torquePedalVariables.TON_torqueOff.IN := FALSE;			// Make sure the torque timer is stopped
	END_IF
	torquePedalVariables.TON_torqueOff();						// Run torque timer
END_ACTION
```

#### LowVoltageBattery.st
```iecst
ACTION LowVoltageBatteryInit:
	lvBatteryConstants.HighLimit := 13.0;
	lvBatteryConstants.LowLimit  := 11.0;

	lvBatteryVariables.TON_batteryEmpty.PT := T#1s;
	lvBatteryVariables.TON_batteryFull.PT := T#1s;
END_ACTION

ACTION LowVoltageBattery:
//	gLowVoltageBattery.data.lowVoltageBatteryVoltage :=  0.001209 * gLowVoltageBattery.inputs.im_LowVoltageBattery_Voltage + 0.6351;
	gLowVoltageBattery.data.voltage :=  (32.0/32767.0) * gLowVoltageBattery.inputs.ai_voltage;

	gLowVoltageBattery.data.current := (((10.0/32767.0)*gLowVoltageBattery.inputs.ai_current) - 0.5)/0.08;

	// Check if the low voltage battery is below a threshold and set status flag
	lvBatteryVariables.TON_batteryEmpty(IN := gLowVoltageBattery.data.voltage < lvBatteryConstants.LowLimit);
	gLowVoltageBattery.status.empty := lvBatteryVariables.TON_batteryEmpty.Q;

	// Check of the low voltage battery is above a threshold and set status flag
	lvBatteryVariables.TON_batteryFull(IN := gLowVoltageBattery.data.voltage > lvBatteryConstants.HighLimit);
	gLowVoltageBattery.status.full := lvBatteryVariables.TON_batteryFull.Q;

END_ACTION
```

### globalSensorNet.var
```iecst
VAR
	gSensorNet : gSensorNet_typ;
END_VAR
VAR CONSTANT
	SENSOR_NET_POLY_LEN : USINT := 8; (*Length - 1. Writing 8 here means its a 9th order polynomial*)
END_VAR
```

### Program Logical/SensorNet/globalSensorNet

#### Main.st
```iecst
PROGRAM _INIT
	(* Insert code here *)

END_PROGRAM

PROGRAM _CYCLIC

	calculateSensorNetOut_0(input := gSensorNet.data.coolingTemp1.input, polyCoeffs := gSensorNet.data.coolingTemp1.polyCoeffs);
	gSensorNet.data.coolingTemp1.value := calculateSensorNetOut_0.output;

END_PROGRAM

PROGRAM _EXIT
	(* Insert code here *)

END_PROGRAM
```

### globalRTDS.var
```iecst
VAR
	gRTDS : gRTDS_typ;
END_VAR
```

### Program Logical/Actuators/Output (IEC)

#### Types.typ - Local data types
```iecst
TYPE
	rtdsVariables_typ : 	STRUCT
		TON_RTDS : TON;
	END_STRUCT;
	rtdsConstants_typ : 	STRUCT
		RTDSCurrent : INT;
	END_STRUCT;
END_TYPE
```

#### Variables.var - Local variables
```iecst
VAR
	i : USINT;
	rtdsVariables : rtdsVariables_typ;
	rtdsConstants : rtdsConstants_typ;
END_VAR
```

### globalCooling.typ
```iecst
TYPE
	gCooling_typ : 	STRUCT
		outputs : gCooling_outputs_typ;
		inputs : gCooling_inputs_typ;
		data : gCooling_data_typ;
		cmd : gCooling_cmd_typ;
		status : gCooling_status_typ;
	END_STRUCT;
	gCooling_outputs_typ : 	STRUCT
		do_fan : ARRAY[0..NUMBER_OF_FANS]OF BOOL;
		do_pump : ARRAY[0..NUMBER_OF_PUMPS]OF BOOL;
	END_STRUCT;
	gCooling_inputs_typ : 	STRUCT
		ai_coolingTemp : ARRAY[0..NUMBER_OF_COOLING_SENSORS]OF INT;
		im_pumpCurrent : ARRAY[0..NUMBER_OF_PUMPS]OF INT;
	END_STRUCT;
	gCooling_cmd_typ : 	STRUCT
		manualMode : BOOL;
		inverterMaxTemp : REAL;
		motorMaxTemp : REAL;
	END_STRUCT;
	gCooling_status_typ : 	STRUCT
		ok : BOOL;
		error : BOOL;
		pumpError : ARRAY[0..1]OF BOOL;
		pumpState : ARRAY[0..1]OF PUMP_STATES;
		warningHighTemperature : BOOL;
		warningInverterHighTemp : BOOL;
		warningMotorHighTemp : BOOL;
	END_STRUCT;
	gCooling_data_typ : 	STRUCT
		coolingSysTemp : ARRAY[0..NUMBER_OF_COOLING_SENSORS]OF REAL;
	END_STRUCT;
	PUMP_STATES :
		(
		PUMP_STATE_OK,
		PUMP_STATE_NO_WATER,
		PUMP_STATE_NOT_CONNECTED
		);
END_TYPE
```

### globalCooling.var
```iecst
VAR CONSTANT
	NUMBER_OF_FANS : USINT := 2;
	NUMBER_OF_COOLING_SENSORS : USINT := 2;
	NUMBER_OF_PUMPS : USINT := 2;
END_VAR
VAR
	gCooling : gCooling_typ;
END_VAR
```

### globalINS.typ
```iecst
TYPE
	gINS_status_typ : 	STRUCT
		ok : BOOL;
	END_STRUCT;
	gINS_data_typ : 	STRUCT
		actLonVelocity_ms : REAL;
		actLatVelocity_ms : REAL;
		actLonVelocity_kmh : REAL;
		actLatVelocity_kmh : REAL;
		actLonAcceleration : REAL;
		actLatAcceleration : REAL;
		actYawRate : REAL;
		actDistTraveledKm : REAL;
		actDistTraveledM : REAL;
		distEstimated : REAL;
	END_STRUCT;
	gINS_input_typ : 	STRUCT
		gyroX : REAL;
		gyroY : REAL;
		gyroZ : REAL;
		accX : REAL;
		accY : REAL;
		accZ : REAL;
		velX : REAL;
		velY : REAL;
		velZ : REAL;
	END_STRUCT;
	gINS_typ : 	STRUCT
		data : gINS_data_typ;
		status : gINS_status_typ;
		input : gINS_input_typ;
	END_STRUCT;
END_TYPE
```

### Program Logical/INS/INS (IEC)

#### Variables.var - Local variables
```iecst
VAR
	messageOk : BOOL;
	distDelta : REAL;
	cycletime : UDINT;
	RTInfo_0 : RTInfo;
	Receiver : Receiver_typ := (0); (*local Struktur with all instances and variables*)
END_VAR
VAR CONSTANT
	BUSY : UINT := 65535; (*Functionblock BUSY status*)
END_VAR
VAR
	socActual : REAL;
	socPrevious : REAL;
	distActual : REAL;
	distPrevious : REAL;
	MTFilterMovingAverage_0 : MTFilterMovingAverage;
	TON_rangEstTimer : TON;
END_VAR
```

#### extractInsData.st
```iecst
(* Action to pick out data for each variable from the received INS data *)
ACTION extractInsData:

	// Byte 0-5: Header

	// Data

	// 6 - 9: AccX
	memcpy(ADR(gINS.input.accX), ADR(Receiver.receive_data)+6,4);
	// 10-13: AccY
	memcpy(ADR(gINS.input.accY), ADR(Receiver.receive_data)+10,4);
	// 14-17: AccZ
	memcpy(ADR(gINS.input.accZ), ADR(Receiver.receive_data)+14,4);

	// 18-21: GyroX
	memcpy(ADR(gINS.input.gyroX), ADR(Receiver.receive_data)+18,4);
	// 22-25: GyroY
	memcpy(ADR(gINS.input.gyroY), ADR(Receiver.receive_data)+22,4);
	// 26-29: GyroZ
	memcpy(ADR(gINS.input.gyroZ), ADR(Receiver.receive_data)+26,4);

	// 30-33: VelX
	memcpy(ADR(gINS.input.velX), ADR(Receiver.receive_data)+30,4);
	// 34-37: VelY
	memcpy(ADR(gINS.input.velY), ADR(Receiver.receive_data)+34,4);
	// 38-41: VelZ
	memcpy(ADR(gINS.input.velZ), ADR(Receiver.receive_data)+38,4);

	// 42-42: Checksum / CRC

END_ACTION
```

#### rangeEst.st
```iecst
ACTION rangeEstimation:
	(* Handle timer *)
	TON_rangEstTimer.IN := TRUE;
	TON_rangEstTimer();

	socActual 	:= gAMS.data.stateOfCharge;
	distActual 	:= gINS.data.actDistTraveledKm;

	(* If timeout occurs *)
	IF TON_rangEstTimer.Q THEN
		(* Reset Timer *)
		TON_rangEstTimer(IN := FALSE);
		(* if the previous SoC is higher *)
		IF socActual < socPrevious THEN
			(* Calculate next value in range estimation *)
			MTFilterMovingAverage_0(In := LIMIT(0,distPrevious - (socPrevious*(distActual-distPrevious))/(socActual-socPrevious),50));
			gINS.data.distEstimated := MTFilterMovingAverage_0.Out;
			(* Previous SoC is lower than new, indication of charging *)
		END_IF;
		distPrevious := gINS.data.actDistTraveledKm;
		socPrevious  := gAMS.data.stateOfCharge;
	END_IF;
END_ACTION
```

#### distMeas.st
```iecst
ACTION distanceMeasurement:

	// dt = cycletime
	// h = ms/(1000*60*60) => h = ms/(3600000)
	distDelta := gINS.data.actLonVelocity_kmh * (UDINT_TO_REAL(cycletime)/3600000.0);

	// Increment distance traveled by distance delta
	gINS.data.actDistTraveledKm := gINS.data.actDistTraveledKm + distDelta;

	// Calculate the distance in meters as well
	gINS.data.actDistTraveledM := gINS.data.actDistTraveledKm*1000.0;

END_ACTION
```

#### checkMessageValidity.st
```iecst
ACTION checkMessageValidity:
	messageOk := TRUE;
END_ACTION
```

### Program Logical/Misc/DataLogging/DataLog

#### Types.typ
```iecst
TYPE
	this_typ : 	STRUCT
		state : UINT;
		tmpStr : STRING[80];
		idxStr : STRING[10];
		strIdxPos : DINT;
		csvData : ARRAY[0..DATALOG_MAX_LOG_VARS]OF STRING[200];
		fileInfoSetting : fiFILE_INFO;
		DTGetTime_0 : DTGetTime;
		header : MpRecipeXmlHeaderType;
		MpDataRegPar : ARRAY[0..DATALOG_MAX_MAPP_VARS]OF MpDataRegPar;
		timestamp : this_timestamp_typ;
		pvData : ARRAY[0..DATALOG_MAX_LOG_VARS]OF this_pvdata_typ;
		pvRegData : ARRAY[0..DATALOG_MAX_MAPP_VARS]OF this_pvRegData_typ;
		okToRestart : BOOL;
		TON_errorReset : TON;
		TON_recordDelay : TON;
		systemReadyToLog : BOOL;
		maxIdxVariableX : USINT;
		brdkUSBConnect_0 : brdkUSBConnect;
		FileCreate_0 : FileCreate;
	END_STRUCT;
	this_timestamp_typ : 	STRUCT
		str : STRING[64];
		old : DATE_AND_TIME;
	END_STRUCT;
	this_pvdata_typ : 	STRUCT
		variable : STRING[200];
		enableVar : STRING[200];
	END_STRUCT;
	this_pvRegData_typ : 	STRUCT
		variable : STRING[100];
		enableVar : STRING[100];
		enable : BOOL;
		address : UDINT;
		datalength : UDINT;
	END_STRUCT;
END_TYPE
```

#### Variables.var
```iecst
VAR
	this : this_typ;
	i : UINT;
	j : USINT;
	pBool : REFERENCE TO BOOL; (*Temp pointer to bool*)
	noOfPvVars : UINT;
	MpDataRecorder_0 : MpDataRecorder;
	MpDataRecorderConfig_0 : MpDataRecorderConfig;
	MpDataRecorderConfiguration : MpDataRecorderConfigType;
	MpRecipeCsv_0 : MpRecipeCsv;
	MpRecipeRegPar_csv : MpRecipeRegPar;
	FileInfo_0 : FileInfo;
	DirCreate_0 : DirCreate;
	RTInfo_0 : RTInfo;
END_VAR
```

#### DataLog.st
```iecst
PROGRAM _INIT

	RTInfo_0(enable := TRUE);
	initSetup;

END_PROGRAM

PROGRAM _CYCLIC
	// call actions
	setup;

	//detect if config.enable is changed then restart datalog
	FOR i:=0 TO DATALOG_MAX_MAPP_VARS DO
		IF this.okToRestart AND this.pvRegData[i].variable <> '' THEN
			IF this.pvRegData[i].address <> 0 AND this.pvRegData[i].datalength = 1 THEN
				pBool ACCESS this.pvRegData[i].address;
				IF pBool <> this.pvRegData[i].enable THEN
					this.state := 0; //restart
				END_IF
			END_IF
		ELSE EXIT;
		END_IF
	END_FOR

	//if file is changed then restart datalog
	FileInfo_0();
	IF this.okToRestart AND this.timestamp.old <> this.fileInfoSetting.modTime THEN
		this.state := 0; //restart
	END_IF

	CASE this.state OF
		0:	// wait for connected usb device
			IF this.brdkUSBConnect_0.status = BRDK_USB_STATUS_FB_READY THEN
				// finds the first available node
				FOR i := 0 TO BRDK_USB_MAX_DEVICES-1 DO
					IF this.brdkUSBConnect_0.node[i].device <> '' THEN
						this.FileCreate_0.pDevice	:= ADR(this.brdkUSBConnect_0.node[i].device);
						this.state := 5;
					END_IF
				END_FOR
			END_IF

		5: //create log folder
			this.okToRestart := FALSE;
			this.timestamp.old := this.fileInfoSetting.modTime;
			MpDataRecorder_0.Enable := FALSE;
			DirCreate_0.enable := TRUE;
			IF DirCreate_0.status = fiERR_DIR_ALREADY_EXIST THEN
				DirCreate_0.enable := FALSE;
				this.state := 10;
			END_IF
			DirCreate_0();

		10:
			MpRecipeRegPar_csv.Enable := TRUE;
			IF MpRecipeRegPar_csv.Active THEN
				this.state := 20;
			ELSIF MpRecipeRegPar_csv.Error THEN
				this.state := 65000;
			END_IF

		20:
			MpRecipeCsv_0.Enable := TRUE;
			IF MpRecipeCsv_0.Active THEN
				this.state := 30;
			ELSIF MpRecipeCsv_0.Error THEN
				this.state := 65000;
			END_IF

		30: //DatalogSettings.csv ok?
			IF FileInfo_0.status = ERR_OK THEN
				this.state := 40;
			ELSIF FileInfo_0.status = fiERR_FILE_NOT_FOUND THEN
				this.state := 300;
			ELSIF FileInfo_0.status = ERR_FUB_BUSY THEN
			ELSE
				this.state := 65000;
			END_IF

		40:
			MpRecipeCsv_0.Load := TRUE;
			IF MpRecipeCsv_0.CommandDone THEN
				MpRecipeCsv_0.Load := FALSE;
				this.state := 45;
			ELSIF MpRecipeCsv_0.Error THEN
				this.state := 65000;
			END_IF

		45:
			MpDataRecorder_0.Enable := TRUE;
			IF MpDataRecorder_0.Active THEN
				this.state := 50;
			ELSIF MpDataRecorder_0.Error THEN
				this.state := 65000;
			END_IF

		50://find logVar#logVarEnable and split it
			brsmemset(ADR(this.pvRegData), 0, SIZEOF(this.pvRegData));
			brsmemset(ADR(this.pvData), 0, SIZEOF(this.pvData));
			FOR i:=0 TO DATALOG_MAX_LOG_VARS DO
				IF gDataLogging.data.csvData[i] <> '' THEN
					this.strIdxPos := brdkStrSearch(ADR(gDataLogging.data.csvData[i]),ADR('#'));
					IF this.strIdxPos > 0 THEN //enable/disable variable found
						this.pvData[i].variable 	:= gDataLogging.data.csvData[i];
						this.pvData[i].enableVar 	:= gDataLogging.data.csvData[i];
						brdkStrSlice(ADR(this.pvData[i].variable), 0, this.strIdxPos);
						brdkStrSlice(ADR(this.pvData[i].enableVar), this.strIdxPos+1, SIZEOF(this.pvData[i].enableVar));
					ELSE
						this.pvData[i].variable := gDataLogging.data.csvData[i];
					END_IF
				ELSE EXIT;
				END_IF
			END_FOR
			this.state := 60;

		60://find and replace [x]. to [0..this.maxIdxVariableX]
			noOfPvVars := 0;
			FOR i:=0 TO DATALOG_MAX_LOG_VARS DO
				IF gDataLogging.data.csvData[i] <> '' THEN
					this.strIdxPos := brdkStrSearch(ADR(this.pvData[i].variable), ADR('[x]'));
				 	IF this.strIdxPos > 0 THEN
				 		FOR j:=0 TO this.maxIdxVariableX DO
							this.tmpStr := '[x]';
							brsitoa(j, ADR(this.idxStr));
							brdkStrReplace(ADR(this.tmpStr), ADR('x'), ADR(this.idxStr));
							this.pvRegData[noOfPvVars].variable 	:= this.pvData[i].variable;
							this.pvRegData[noOfPvVars].enableVar 	:= this.pvData[i].enableVar;
							brdkStrReplace(ADR(this.pvRegData[noOfPvVars].variable), ADR('[x]'), ADR(this.tmpStr));
							brdkStrReplace(ADR(this.pvRegData[noOfPvVars].enableVar), ADR('[x]'), ADR(this.tmpStr));
							PV_xgetadr(ADR(this.pvRegData[noOfPvVars].enableVar), ADR(this.pvRegData[noOfPvVars].address), ADR(this.pvRegData[noOfPvVars].datalength));
							noOfPvVars := noOfPvVars + 1;
						END_FOR
					ELSE
						this.pvRegData[noOfPvVars].variable 	:= this.pvData[i].variable;
						this.pvRegData[noOfPvVars].enableVar 	:= this.pvData[i].enableVar;
						PV_xgetadr(ADR(this.pvRegData[noOfPvVars].enableVar), ADR(this.pvRegData[noOfPvVars].address), ADR(this.pvRegData[noOfPvVars].datalength));
						noOfPvVars := noOfPvVars + 1;
				 	END_IF
				ELSE EXIT;
				END_IF
			END_FOR
			this.state := 65;

		65: //clear all reg pars before init again
			FOR i:=0 TO DATALOG_MAX_MAPP_VARS DO
				this.MpDataRegPar[i].Enable := FALSE;
			END_FOR
			this.state := 70;

		70: //registre pv's
			FOR i:=0 TO DATALOG_MAX_MAPP_VARS DO
				IF this.pvRegData[i].variable <> '' THEN
					this.MpDataRegPar[i].MpLink 		:= ADR(gDataRecorder);
					this.MpDataRegPar[i].Description 	:= ADR(this.pvRegData[i].variable);
					this.MpDataRegPar[i].PVName			:= ADR(this.pvRegData[i].variable);
					IF this.pvRegData[i].address <> 0 AND this.pvRegData[i].datalength = 1 THEN
						pBool ACCESS this.pvRegData[i].address;
						this.pvRegData[i].enable := pBool;
					ELSE
						this.pvRegData[i].enable := TRUE;
					END_IF
					this.MpDataRegPar[i].Enable	:= this.pvRegData[i].enable;
				ELSE EXIT;
				END_IF
			END_FOR
			this.okToRestart := TRUE;
			this.state := 80;

		80: //wait for system up and running
			IF this.systemReadyToLog THEN
				MpDataRecorder_0.Enable := TRUE;
				this.state := 85;
			END_IF

		85: //active
			IF MpDataRecorder_0.Active THEN
				this.TON_recordDelay.IN := TRUE;
				this.state := 90;
			ELSIF MpDataRecorder_0.Error THEN
				this.state := 65000;
			END_IF

		90: //delay before start recording
			IF this.TON_recordDelay.Q THEN
				this.TON_recordDelay.IN := FALSE;
				MpDataRecorder_0.Record := TRUE;
				this.state := 100;
			END_IF

		100: //ready
			gDataLogging.status.dataloggingActive := TRUE;
			IF gCreateLogFile THEN
				this.okToRestart := FALSE;
				MpDataRecorder_0.SnapShot := TRUE;
				this.state := 110;
			ELSIF NOT MpDataRecorder_0.Enable THEN // restart after download
				gCreateLogFile := FALSE;
				this.state := 0;
			ELSIF MpDataRecorder_0.Error THEN
				gCreateLogFile := FALSE;
				this.state := 65000;
			END_IF

			IF MpDataRecorder_0.Info.CurrentFileSize > 900 THEN
				this.state := 5;
			END_IF

		110: //waiting for datalog file created
			IF MpDataRecorder_0.SnapShotDone THEN
				MpDataRecorder_0.SnapShot 	:= FALSE;
				gCreateLogFile 				:= FALSE;
				this.state 					:= 100;
			ELSIF MpDataRecorder_0.Error THEN
				MpDataRecorder_0.ErrorReset	:= TRUE;
				MpDataRecorder_0.SnapShot 	:= FALSE;
				gCreateLogFile 				:= FALSE;
				this.state 					:= 65000;
			END_IF

		300: //create DatalogSettings.csv
			MpRecipeCsv_0.Save := TRUE;
			IF MpRecipeCsv_0.CommandDone THEN
				MpRecipeCsv_0.Save := FALSE;
				this.state := 0;
			ELSIF MpRecipeCsv_0.Error THEN
				this.state := 65000;
			END_IF

		65000://ERROR HANDLING = NONE :/
			this.TON_errorReset.IN	:= TRUE;
			IF this.TON_errorReset.Q THEN
				this.TON_errorReset.IN		:= FALSE;
				MpDataRecorder_0.Enable 	:= FALSE;
				MpRecipeRegPar_csv.Enable 	:= FALSE;
				MpRecipeCsv_0.Enable		:= FALSE;
				FileInfo_0.enable			:= FALSE;
				this.state					:= 0;
			END_IF

	END_CASE

	// Function Block Calls
	this.TON_errorReset(PT := T#10s);

	IF this.state <> 100 OR this.brdkUSBConnect_0.status <> BRDK_USB_STATUS_FB_READY THEN
		gDataLogging.status.dataloggingActive := FALSE;
	END_IF

	this.TON_recordDelay();
	IF MpDataRecorder_0.Active THEN
		FOR i:=0 TO DATALOG_MAX_MAPP_VARS DO
			this.MpDataRegPar[i]();
		END_FOR
	END_IF
	MpDataRecorderConfig_0();
	MpDataRecorder_0();
	MpRecipeRegPar_csv();
	MpRecipeCsv_0();
	this.brdkUSBConnect_0();

END_PROGRAM

PROGRAM _EXIT
	// Disable Mapp Function Blocks
	MpDataRecorder_0(Enable := FALSE);
	MpDataRecorderConfig_0(Enable := FALSE);
	MpRecipeCsv_0(Enable := FALSE);
	MpRecipeRegPar_csv(Enable := FALSE);
END_PROGRAM
```

#### setup.st
```iecst
ACTION setup:
	IF this.brdkUSBConnect_0.node[0].device <> '' THEN
		MpRecipeRegPar_csv.MpLink 	:= ADR(gRecipeCsv);
		MpRecipeRegPar_csv.PVName 	:= ADR('DataLog:gDataLogging.inputs.csvData');
		MpRecipeRegPar_csv.Category	:= ADR('datalogSettings');

		MpRecipeCsv_0.MpLink 		:= ADR(gRecipeCsv);
		MpRecipeCsv_0.DeviceName 	:= ADR(this.brdkUSBConnect_0.node[0].device);
		MpRecipeCsv_0.FileName 		:= ADR('log/DatalogSettings');
		MpRecipeCsv_0.Category		:= ADR('datalogSettings');

		MpDataRecorder_0.MpLink			:= ADR(gDataRecorder);
		MpDataRecorder_0.DeviceName		:= ADR(this.brdkUSBConnect_0.node[0].device);
		MpDataRecorder_0.RecordMode 	:= mpDATA_RECORD_MODE_TIME;
		MpDataRecorder_0.SamplingTime	:= RTInfo_0.cycle_time / 1000; //micro to milli

		MpDataRecorderConfiguration.DecimalDigits	:= 3;
		MpDataRecorderConfiguration.BufferSize		:= 50000; //kB
		MpDataRecorderConfiguration.PowerFailSafe	:= FALSE;
		MpDataRecorderConfiguration.FileNamePattern	:= 'Datalog_%Y%m%d_%H%M%S.csv';
		MpDataRecorderConfiguration.DecimalMark		:= '.';
		MpDataRecorderConfiguration.AutoSave		:= FALSE;

		MpDataRecorderConfig_0.MpLink 				:= ADR(gDataRecorder);
		MpDataRecorderConfig_0.Configuration		:= ADR(MpDataRecorderConfiguration);
		MpDataRecorderConfig_0.Enable 				:= TRUE;

		FileInfo_0.pDevice			:= ADR(this.brdkUSBConnect_0.node[0].device);
		FileInfo_0.pName			:= ADR('log/DatalogSettings.csv');
		FileInfo_0.pInfo			:= ADR(this.fileInfoSetting);
		FileInfo_0.enable			:= TRUE;

		DirCreate_0.pDevice			:= ADR(this.brdkUSBConnect_0.node[0].device);
		DirCreate_0.pName			:= ADR('log');

		this.TON_recordDelay.PT 	:= T#10ms;
		this.maxIdxVariableX 		:= 0;
		this.systemReadyToLog 		:= TRUE;
	END_IF
END_ACTION
```

### Program Logical/Misc/DataLogging/sampleST (IEC)

#### Cyclic.st - Cyclic code
```iecst
PROGRAM _INIT

	this.fileName 	:= 'brdkUSB.txt';
	this.fileSource := 'brdkUSB is a great library';

END_PROGRAM

PROGRAM _CYCLIC

	CASE this.state OF

		0:	// wait for connected usb device
			IF this.brdkUSBConnect_0.status = BRDK_USB_STATUS_FB_READY THEN
				// finds the first avaible node
				FOR i := 0 TO BRDK_USB_MAX_DEVICES-1 DO
					IF this.brdkUSBConnect_0.node[i].device <> '' THEN
						this.FileCreate_0.pDevice	:= ADR(this.brdkUSBConnect_0.node[i].device);
						this.state := 10;
					END_IF
				END_FOR

			END_IF

		10:	// wait for command
			IF this.brdkUSBConnect_0.status = BRDK_USB_STATUS_FB_READY THEN
				IF this.cmd.createFile THEN
					this.cmd.createFile 		:= FALSE;
					this.FileCreate_0.enable 	:= TRUE;
					this.FileCreate_0.pFile		:= ADR(this.fileName);
					this.FileCreate_0();
					this.state := 20;
				END_IF
			ELSE
				this.state := 0;
			END_IF

		20:	// wait for file to be created on usb device
			this.FileCreate_0();
			CASE this.FileCreate_0.status OF

				ERR_OK:
					this.FileWrite_0.enable := TRUE;
					this.FileWrite_0.ident 	:= this.FileCreate_0.ident;
					this.FileWrite_0.offset := 0;
					this.FileWrite_0.pSrc 	:= ADR(this.fileSource);
					this.FileWrite_0.len	:= brsstrlen(ADR(this.fileSource));
					this.state 				:= 40;

				fiERR_EXIST:
					this.FileDelete_0.enable 	:= TRUE;
					this.FileDelete_0.pDevice 	:= this.FileCreate_0.pDevice;
					this.FileDelete_0.pName 	:= this.FileCreate_0.pFile;
					this.FileDelete_0();
					this.state 					:= 30;

			END_CASE

		30:	// delete file if it already exists
			this.FileDelete_0();
			CASE this.FileDelete_0.status OF

				ERR_OK,fiERR_FILE_NOT_FOUND:
					this.cmd.createFile := TRUE;
					this.state 			:= 10;

			END_CASE

		40:	// write to file
			this.FileWrite_0();
			CASE this.FileWrite_0.status OF

				ERR_OK:
					this.FileClose_0.enable := TRUE;
					this.FileClose_0.ident 	:= this.FileCreate_0.ident;
					this.FileClose_0();
					this.state := 50;

			END_CASE

		50:	// wait for file to be closed
			this.FileClose_0();
			CASE this.FileClose_0.status OF

				ERR_OK,fiERR_FILE_NOT_OPENED:
					this.state := 10;

			END_CASE

	END_CASE

	this.brdkUSBConnect_0();

END_PROGRAM
```

#### Types.typ - Local data types
```iecst
TYPE
	brdkusb_sample_st_cmd_typ : 	STRUCT
		createFile : BOOL;
	END_STRUCT;
	brdkusb_sample_st_interal_typ : 	STRUCT
		state : UINT;
		brdkUSBConnect_0 : brdkUSBConnect;
		cmd : brdkusb_sample_st_cmd_typ;
		FileCreate_0 : FileCreate;
		FileClose_0 : FileClose;
		FileWrite_0 : FileWrite;
		FileDelete_0 : FileDelete;
		fileName : STRING[80];
		fileSource : STRING[100];
	END_STRUCT;
END_TYPE
```

- Visualisation Logical/mappView (not shown)

Listed in the project but not available here: Logical/Global.var, Logical/SM/StateMachine/Main.st, Logical/SM/StateMachine/Variables.var, Logical/SM/StateMachine/states/stateIdle.st, Logical/SM/StateMachine/states/stateSCEnabled.st, Logical/SM/StateMachine/states/statePrecharging.st, Logical/SM/StateMachine/states/stateTractive.st, Logical/SM/StateMachine/states/stateDrive.st, Logical/SM/StateMachine/states/stateError.st, Logical/SM/StateMachine/functions/instruction.st, Logical/Inverters/CAN/CAN/Main.st, Logical/Inverters/CAN/CAN/Types.typ, Logical/Inverters/CAN/CAN/Variables.var, Logical/Inverters/Control/Control/Variables.var, Logical/Inverters/Control/Control/Controllers/powerLimiter.st, Logical/Inverters/Control/Control/Controllers/regenerativeBraking.st, Logical/Inverters/Inv_statemachine/Inv_statemachine/hmiAction.st, Logical/Inverters/Inv_statemachine/Inv_statemachine/mission.st, Logical/AMS_and_Shunt/AMS/Main.st, Logical/AMS_and_Shunt/AMS/Variables.var, Logical/AMS_and_Shunt/AMS/powerMonitoring.st, Logical/AMS_and_Shunt/AMS/eventLog, Logical/AMS_and_Shunt/CAN/AMS_CAN/Main.st, Logical/AMS_and_Shunt/CAN/AMS_CAN/Types.typ, Logical/Dashboard/globalDashboard.var, Logical/Dashboard/Dashboard/Main.st, Logical/Dashboard/Dashboard/errors.st, Logical/Dashboard/Dashboard/can.st, Logical/Dashboard/Dashboard/Receive/Receive_Bus.st, Logical/Dashboard/Dashboard/Receive/receive_messages.st, Logical/Dashboard/Dashboard/ErrorDashboard.st, Logical/Dashboard/Dashboard/eventLog, Logical/Sensors/globalSteeringAngle.typ, Logical/Sensors/globalSteeringAngle.var, Logical/Sensors/globalBraking.typ, Logical/Sensors/globalBraking.var, Logical/Sensors/globalTorqueSensor.var, Logical/Sensors/Sensors/Main.st, Logical/Sensors/Sensors/Variables.var, Logical/Sensors/Sensors/SteeringAngle, Logical/Actuators/globalRTDS.typ, Logical/Actuators/Output/Main.st, Logical/Actuators/Output/RTDS/RTDS.st, Logical/CoolingSystem/COOLING, Logical/INS/globalINS.var, Logical/INS/INS/Main.st, Logical/INS/INS/Types.typ, Logical/Misc/AlarmManagement/AlarmManagement, Logical/Misc/DataLogging/sampleST/Variables.var
